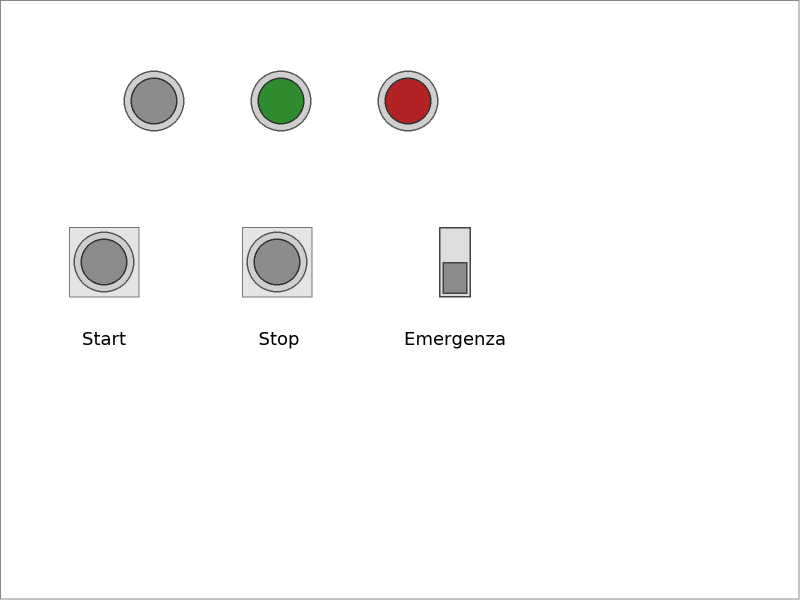
VISUALIZATION Visualization  // 800x600
    Label (29,324 150x30), "Start"
    Lamp1 (119,66 70x70), variable: GVL.MachineIsActive, style: Lamp-Lamp1-Gray
    Lamp1 (246,66 70x70), variable: GVL.MachineIsRunning, style: Lamp-Lamp1-Green
    Lamp1 (373,66 70x70), variable: GVL.Emergency, style: Lamp-Lamp1-Red
    PushSwitch (69,227 70x70), variable: GVL.PBStart, behaviour: TAP, style: Switch-PushSwitch-Gray
    Label (204,324 150x30), "Stop"
    PushSwitch (242,227 70x70), variable: GVL.PBStop, behaviour: TAP, style: Switch-PushSwitch-Gray
    DipSwitch (420,227 70x70), variable: GVL.PBEmergency, behaviour: TOGGLE, style: Switch-DipSwitch-Gray
    Label (380,324 150x30), "Emergenza"
END_VISUALIZATION

(* stored: Version 1.1.0.1, ProductVersion 3.1.4024.12
   Visu Visualization: Id {e1523be8-0b27-41d4-ac07-354f31b26bca} *)
